TYPE ST_SP_ProcessCmd :
STRUCT
	rMixerSpeed				:REAL;
	bMixerStart				:BOOL;
	rHeaterTemperature		:REAL;
	bHeaterStart			:BOOL;
END_STRUCT
END_TYPE

(* stored: Version 1.1.0.1, ProductVersion 3.1.4024.12
   DUT ST_SP_ProcessCmd: Id {f1683f0a-438a-4d14-b04b-1aa42e747844} *)
